_CFC_ (* Continuous Function Chart, elements in execution order *)
#0 TON_sost_VKL:TON(IN: SCHU_P2_2_UST_SOST_VKL, PT: T#500ms)
#1 OR(SCHU_P2_2_M1_B45, SCHU_P2_2_M2_B45)
#2 RT_VKL:R_TRIG(CLK: #0.Q)
#3 AND(#2.Q, NOT SCHU_P2_2_UST_RE_PROGREV)
#4 FT_PROGREV:F_TRIG(CLK: SCHU_P2_2_UST_RE_PROGREV)
#5 OR(#3, #4.Q)
#6 OR(#9, SCHU_P2_2_UST_SOST_OTKL, #11.Q)
#7 RS_Pusk:RS(SET: #5, RESET1: #6)
#8 SCHU_P2_2_UST_RE_PUSK <= #7.Q1
#9 AND(#1, SCHU_P2_2_AVR_A)
#10 AND(SCHU_P2_2_UST_RE_PUSK, SCHU_P2_2_AVR_M)
#11 TON_AVR_M:TON(IN: #10, PT: T#1s)
_END_CFC_
END_PROGRAM

(* POU Regim/Rabota, CFC *)
PROGRAM Rabota
VAR
	RS_Rabota: RS;
	FT_Pusk: F_TRIG;
END_VAR
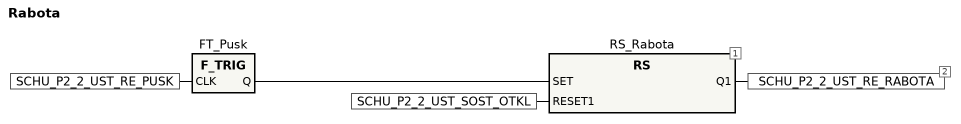
_CFC_ (* Continuous Function Chart, elements in execution order *)
#0 FT_Pusk:F_TRIG(CLK: SCHU_P2_2_UST_RE_PUSK)
#1 RS_Rabota:RS(SET: #0.Q, RESET1: SCHU_P2_2_UST_SOST_OTKL)
#2 SCHU_P2_2_UST_RE_RABOTA <= #1.Q1
_END_CFC_
(* the same logic as Structured Text *)
FT_Pusk(CLK := SCHU_P2_2_UST_RE_PUSK);
RS_Rabota(SET := FT_Pusk.Q, RESET1 := SCHU_P2_2_UST_SOST_OTKL);
SCHU_P2_2_UST_RE_RABOTA := RS_Rabota.Q1;
END_PROGRAM

(* POU IM/ALL_IM, CFC *)
PROGRAM ALL_IM
VAR
END_VAR
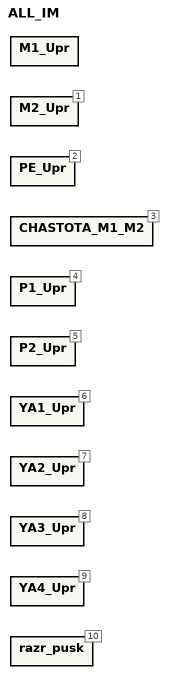
_CFC_ (* Continuous Function Chart, elements in execution order *)
#0 M1_Upr()
#1 M2_Upr()
#2 PE_Upr()
#3 CHASTOTA_M1_M2()
#4 P1_Upr()
#5 P2_Upr()
#6 YA1_Upr()
#7 YA2_Upr()
#8 YA3_Upr()
#9 YA4_Upr()
#10 razr_pusk()
_END_CFC_
(* the same logic as Structured Text *)
M1_Upr();
M2_Upr();
PE_Upr();
CHASTOTA_M1_M2();
P1_Upr();
P2_Upr();
YA1_Upr();
YA2_Upr();
YA3_Upr();
YA4_Upr();
razr_pusk();
END_PROGRAM

(* POU IM/M1_Upr, CFC *)
PROGRAM M1_Upr
VAR
	RS_M1: RS;

	startDelay_M1: TIME := T#0s;
	stopDelay_M1: TIME := T#0s;
	delayFBC_M1: TIME := T#30S;
	feedbPT_M1: TIME := T#120s;
	delayFBP_M1: TIME := T#30s;

	fb_HVACMS_M1: FB_HVACMotor1Speed;
	fb_HVACPIDC_M1: FB_HVACPIDCtrl;

	deadRange: REAL := 0.1;
	rKp: REAL := 1;
	tTi: TIME;
	tTv: TIME := T#0s;
	tTd: TIME := T#0s;
	direction: BOOL;
	rYMin: REAL;
	Dint_Ti: DINT;
	set: BOOL;
	reset: BOOL;
	resetContr: BOOL;
	SR_VKL: SR;
END_VAR
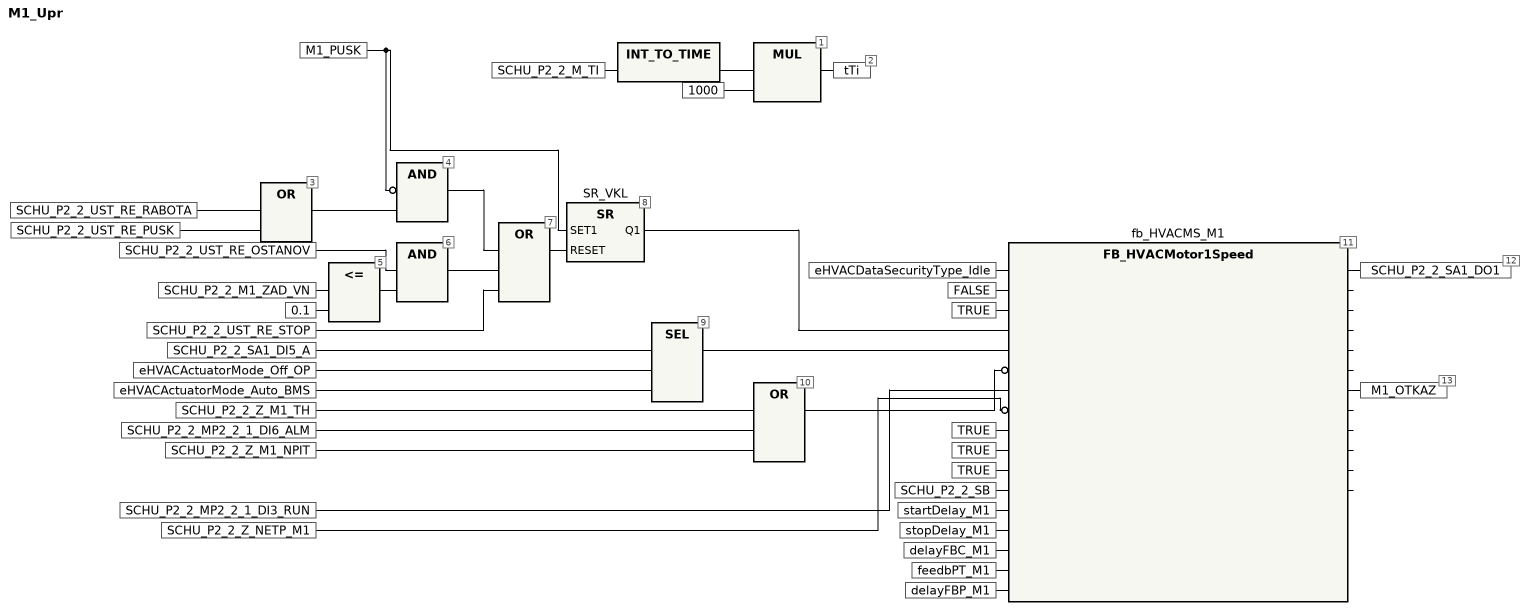
_CFC_ (* Continuous Function Chart, elements in execution order *)
#0 INT_TO_TIME(SCHU_P2_2_M_TI)
#1 MUL(#0, 1000)
#2 tTi <= #1
#3 OR(SCHU_P2_2_UST_RE_RABOTA, SCHU_P2_2_UST_RE_PUSK)
#4 AND(NOT M1_PUSK, #3)
#5 <=(SCHU_P2_2_M1_ZAD_VN, 0.1)
#6 AND(SCHU_P2_2_UST_RE_OSTANOV, #5)
#7 OR(#4, #6, SCHU_P2_2_UST_RE_STOP)
#8 SR_VKL:SR(SET1: M1_PUSK, RESET: #7)
#9 SEL(SCHU_P2_2_SA1_DI5_A, eHVACActuatorMode_Off_OP, eHVACActuatorMode_Auto_BMS)
#10 OR(SCHU_P2_2_Z_M1_TH, SCHU_P2_2_MP2_2_1_DI6_ALM, SCHU_P2_2_Z_M1_NPIT)
#11 fb_HVACMS_M1:FB_HVACMotor1Speed(eHVACDataSecurityType_Idle, FALSE, TRUE, #8.Q1, #9, NOT #10, SCHU_P2_2_MP2_2_1_DI3_RUN, NOT SCHU_P2_2_Z_NETP_M1, TRUE, TRUE, TRUE, SCHU_P2_2_SB, startDelay_M1, stopDelay_M1, delayFBC_M1, feedbPT_M1, delayFBP_M1)
#12 SCHU_P2_2_SA1_DO1 <= #11.out 1
#13 M1_OTKAZ <= #11.out 7
_END_CFC_
END_PROGRAM

(* POU IM/M2_Upr, CFC *)
PROGRAM M2_Upr
VAR
	RS_M2: RS;

	startDelay_M2: TIME := T#0s;
	stopDelay_M2: TIME := T#0s;
	delayFBC_M2: TIME := T#30s;
	feedbPT_M2: TIME := T#120s;
	delayFBP_M2: TIME := T#30s;

	fb_HVACMS_M2: FB_HVACMotor1Speed;
	fb_HVACPIDC_M2: FB_HVACPIDCtrl;

	deadRange: REAL := 0.1;
	rKp: REAL := 1;
	tTi: TIME;
	tTv: TIME := T#0s;
	tTd: TIME := T#0s;
	direction: BOOL;
	rYMin: REAL;
	Dint_Ti: DINT;

	set: BOOL;
	reset: BOOL;
	resetContr: BOOL;
	RR_M2: RAMP_REAL;
	SR_START_REG: SR;
	RT_KOMVKL: R_TRIG;

	speedMotor: REAL;
	SR_VKL: SR;
END_VAR
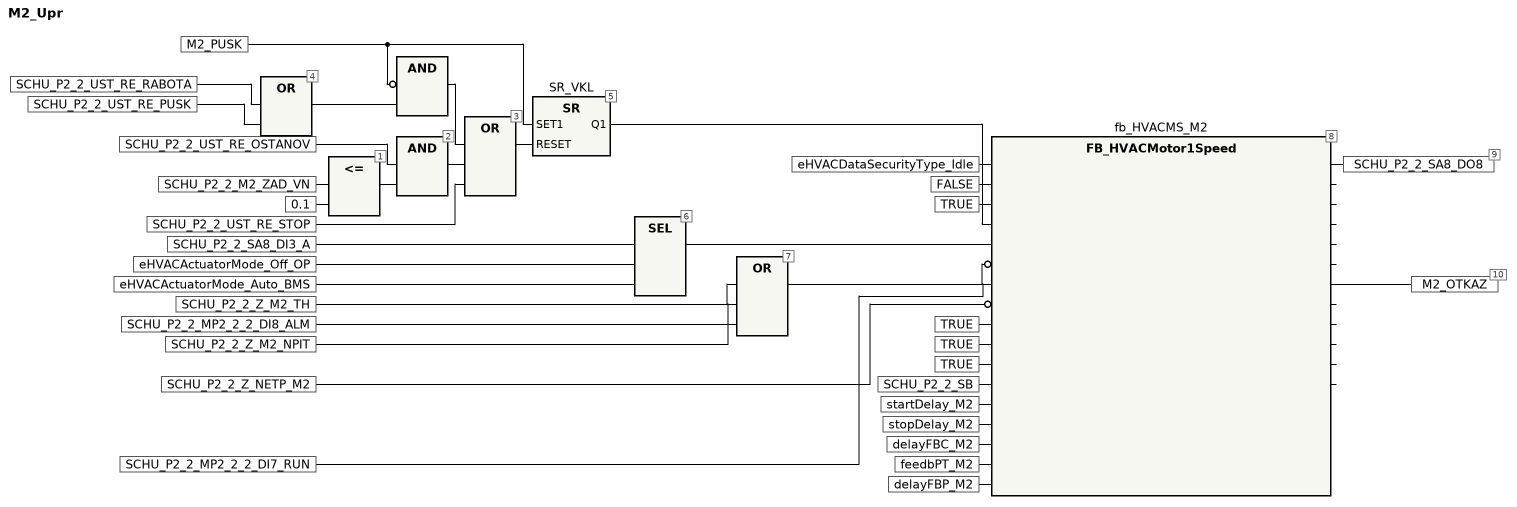
_CFC_ (* Continuous Function Chart, elements in execution order *)
#0 AND(NOT M2_PUSK, #4)
#1 <=(SCHU_P2_2_M2_ZAD_VN, 0.1)
#2 AND(SCHU_P2_2_UST_RE_OSTANOV, #1)
#3 OR(#0, #2, SCHU_P2_2_UST_RE_STOP)
#4 OR(SCHU_P2_2_UST_RE_RABOTA, SCHU_P2_2_UST_RE_PUSK)
#5 SR_VKL:SR(SET1: M2_PUSK, RESET: #3)
#6 SEL(SCHU_P2_2_SA8_DI3_A, eHVACActuatorMode_Off_OP, eHVACActuatorMode_Auto_BMS)
#7 OR(SCHU_P2_2_Z_M2_TH, SCHU_P2_2_MP2_2_2_DI8_ALM, SCHU_P2_2_Z_M2_NPIT)
#8 fb_HVACMS_M2:FB_HVACMotor1Speed(eHVACDataSecurityType_Idle, FALSE, TRUE, #5.Q1, #6, NOT #7, SCHU_P2_2_MP2_2_2_DI7_RUN, NOT SCHU_P2_2_Z_NETP_M2, TRUE, TRUE, TRUE, SCHU_P2_2_SB, startDelay_M2, stopDelay_M2, delayFBC_M2, feedbPT_M2, delayFBP_M2)
#9 SCHU_P2_2_SA8_DO8 <= #8.out 1
#10 M2_OTKAZ <= #8.out 7
_END_CFC_
END_PROGRAM

(* POU IM/PE_Upr, CFC *)
PROGRAM PE_Upr
VAR
	PE_PID: FB_HVACPIDCtrl;

	deadRange: REAL := 0.1;
	direction: BOOL;
	tTi: TIME;
	tTv: TIME;
	tTd: TIME;
	PE_PID_VKL: TON;
END_VAR
